{warning 'Eigenschaftenimplementierung hinzufügen'}
PROPERTY P_SpeedInPercent : LREAL
GET
P_SpeedInPercent := THIS^.rSpeedInPercentToSet;
END_GET
END_PROPERTY

PROPERTY P_StrokeLength : REAL
GET
P_StrokeLength := THIS^.rStrokeLength;
END_GET
END_PROPERTY

{warning 'Eigenschaftenimplementierung hinzufügen'}
PROPERTY P_StrokeLengthInitialized : BOOL
GET
P_StrokeLengthInitialized := THIS^.bStrokeLengthInitialized;
END_GET
SET
THIS^.bStrokeLengthInitialized := P_StrokeLengthInitialized;
END_SET
END_PROPERTY

PROPERTY P_WorkPressure : REAL
GET
P_WorkPressure := THIS^.rCurrentPressureInBar;
END_GET
END_PROPERTY

END_FUNCTION_BLOCK

(* stored: Version 1.1.0.1, ProductVersion 3.1.4024.12
   POU FB_CYLINDER_DA_TESTDEV1: Id {869475c7-ef97-4a7c-8ba5-1a42b23da02a}, SpecialFunc None
   Folder PRIVAT: Id {5831127a-e495-46f5-8a0f-1d046bc33d11}
   Folder SEQUENCE: Id {a9bffe34-56d4-42a0-bd85-2120cfcc493b}
   Method _m_DebugManager: Id {3c0314c9-f958-4098-88b9-d633cb92bde6}
   Method _m_Delay: Id {4de8ce80-6b9e-428f-9ea5-2ff018cbca80}
   Method _m_GeneralStepSetting: Id {24d8fd13-b379-4769-a659-85f3a480beb1}
   Method _m_HMI: Id {f56e0455-8f05-427d-ae10-35ce3dd7ec48}
   Method _m_ManualOperation: Id {08ef6f8c-9fc2-4a0c-ad9f-9f46c3bbc957}
   Method _m_PressureCalibration: Id {34794bd8-8f30-4a1c-bded-6683db0c4b4c}
   Method _m_PressureRegulation: Id {b0e232cf-6ed7-46e2-900f-075612c3a0f9}
   Method _m_Recording: Id {df88b879-7071-4b2f-a597-6e80be8b9c71}
   Method _m_SaveLastStep: Id {9fdaa3b9-a96c-4bff-bb87-77a3e60df6bb}
   Method _m_Seq_INIT: Id {f9cfc93d-4b0f-43dd-ab42-c65811c2e031}
   Method _m_Seq_LOW_PRESSURE_CALIBRATION: Id {1318f128-dd64-4e95-89a0-884e121348f4}
   Method _m_Seq_LOW_PRESSURE_MODE: Id {f82ab1c7-c9ef-435d-9f8b-8c61489859a6}
   Method _m_Seq_OPEN_LOCK_VALVES: Id {b7cfbdb7-7d40-423e-8fff-728fd5186b1e}
   Method _m_Seq_OPEN_RESERVOIR: Id {e1236d95-c6e4-4c6f-a7f3-534cb4bf9b62}
   Method _m_Seq_PRESSURE_CALIBRATION: Id {1bfc6a85-663e-4024-8ab2-022a9e48ea16}
   Method _m_Seq_PUMP2_ADD: Id {1baeb679-c052-4be0-8a42-e0985d7a075e}
   Method _m_Seq_PUMP3_ADD: Id {91b2c056-8d1b-40bd-b9b4-ee7732a8764d}
   Method _m_Seq_PUMP4_ADD: Id {9f51ed93-3bb9-4a3d-8f66-c8bb58c50c06}
   Method _m_Seq_SET_MAX_POS: Id {a4ff45b1-09e0-4222-a355-b456c9816aeb}
   Method _m_Seq_SET_WORK_PRESSURE: Id {cc2c3b1d-434f-4870-918e-924ee5476c2f}
   Method _m_Seq_SET_ZERO_POS: Id {a0698914-5d1c-48f0-b6d0-ead3eebb9680}
   Method _m_Seq_STOP: Id {5a3e320f-112a-4844-b8ff-ad7e993876ce}
   Method _m_Seq_STOP_AND_LOCK: Id {d01e608a-17c4-4d36-a5d6-d8a44fccd4da}
   Method _m_Seq_TO_HP: Id {93cdc5d4-9ecd-488d-babb-0c1575d8e8d4}
   Method _m_Seq_TO_SET_POS: Id {2c0f225f-9b0a-4aae-b925-08b548f42d15}
   Method _m_Seq_TO_WP: Id {5ba5b69d-8d51-4ff0-a3ee-fd4a54b59f89}
   Method _m_SequenceManager: Id {a82c7186-75d7-41f9-a75c-fb34f442338a}
   Method _m_SpeedRegulation: Id {bde6a516-003e-4041-b299-332af2ff0a98}
   Method _m_TimeOut: Id {4d7a21df-4d0e-456e-837a-6e1ec028adba}
   Method FB_init: Id {3eddab45-6958-4dfd-8b24-1deffd8654a6}
   Method M_LowPressureCalibration: Id {4c4aa761-4ce6-4927-99ce-753ef2c83bac}
   Method M_LowPressureMode: Id {ffc0cadb-621c-44b9-8086-c56093a333f6}
   Method M_OpenLockValves: Id {9d7190d5-3e74-4fb9-954e-0504316da3b0}
   Method M_OpenReservoir: Id {4d05e67f-0bcd-4d4d-89ad-643ecfe61b4f}
   Method M_PressureCalibration: Id {95a02b1f-d857-4bb7-8e27-77402689bfbf}
   Method M_Pump2Add: Id {88f3a218-cc95-4bf0-b16d-163da42870b5}
   Method M_Pump3Add: Id {c24a4452-1376-4ce6-a3ab-19c9ec15d08e}
   Method M_Pump4Add: Id {75eda3be-013d-4e3a-b91d-bfd32528cd7a}
   Method M_Reset: Id {51185ceb-0608-4fb2-82ca-2fdc35a10112}
   Method M_Run: Id {23e5959b-1f76-44e9-b254-e7757dbd1b8c}
   Method M_SetMaxPos: Id {bb4d4dca-6123-4524-b431-23bb935eee74}
   Method M_SetReady: Id {d9e65538-b03d-4723-b24c-4503df9eaef2}
   Method M_SetWorkPressure: Id {b51b9fcf-a17a-49ed-b114-876c3efd1a1a}
   Method M_SetZeroPos: Id {3aad99c8-3b93-4b4c-95b9-950170a10e45}
   Method M_Stop: Id {49a98cb3-5742-4c81-97f6-41549c0a6194}
   Method M_StopAndLock: Id {f07563c3-75a4-4012-a26b-70e4e023623a}
   Method M_ToHP: Id {fe8cf06b-e261-4737-851b-dfa0a48b2569}
   Method M_ToSetPos: Id {44cdaf68-bebc-4b53-b732-e3d0c25a0570}
   Method M_ToWP: Id {42eccb49-e3a0-4f84-9df1-89e9492bac4f}
   Property P_ActiveDirection: Id {bb177c56-5bf4-456b-bd35-4110bf2c0b6b}
   Get Get: Id {81862fc7-8740-48d6-aabb-750d3f4aa01e}
   Property P_ActiveVolumeFlow: Id {946f3b6b-b04f-4592-a5d6-37e4a19507d5}
   Get Get: Id {abd0562a-6524-4426-82ad-461c174736ab}
   Property P_CurrentForceInKN: Id {6c649f8a-2cb9-4c53-a460-6728e479212a}
   Get Get: Id {3ee17635-3cb1-47d0-9298-d2a1694411b6}
   Property P_DoubleActing: Id {5d7ac27f-14e0-409a-ba97-dda6248a40da}
   Get Get: Id {0beebe25-6228-4f14-946f-52856e4bb06d}
   Property P_Event: Id {31da0ff1-1dfd-4e32-b8ac-0cb534ab2b59}
   Get Get: Id {ea8eb761-a1fb-4af3-8d9c-dc884b6aba71}
   Set Set: Id {eedfdc11-1201-44c7-91df-13c0241d5659}
   Property P_FullObjectPath: Id {f4b51499-f863-40ce-a072-20999b9fe9a3}
   Get Get: Id {5901c2fa-eda4-4d5d-8c4f-f4141c32c492}
   Set Set: Id {781f8bf3-4ce8-486b-b4b0-51206a6f96d2}
   Property P_Global_Ack: Id {d5036133-64f7-4f9e-a413-2f769fc7f207}
   Get Get: Id {84859d05-d51e-48f0-9b19-2a76ccc49b02}
   Set Set: Id {224b9ca1-1704-4d02-9c9f-2d98b2303f3e}
   Property P_GlobalID: Id {1f8794ac-59f7-4097-9335-26e805a10d87}
   Get Get: Id {0d8c0c77-d0ae-429b-a753-731140411ead}
   Property P_LowPressure: Id {8360123c-b111-49fc-8952-81201de0e957}
   Get Get: Id {f20bbd60-1f27-491c-b237-908a7d58ba07}
   Property P_LowPressureChA: Id {701b8f3f-ea17-4898-9856-3b520b81dd7e}
   Get Get: Id {ecdb97ab-3f8e-4a79-b663-74b2d1833e48}
   Property P_LowPressureChB: Id {8572c222-9080-4ca7-880d-9909692f2624}
   Get Get: Id {728077ee-e2ba-4ef8-99a2-da95007fc54c}
   Property P_LowPressureModeEnable: Id {1fe6839d-8940-4533-a401-c4cc583e6577}
   Get Get: Id {4e27dfa8-7aa6-4726-8e1e-1c44da369649}
   Property P_MaxPosVal: Id {cff043fe-ab6a-47f5-aa1a-c070fe6ac24e}
   Get Get: Id {c5fbf8f1-9ff5-46c4-aa5d-f85bafebb367}
   Property P_MinPosVal: Id {be0fed34-5310-407d-9569-733869df6eed}
   Get Get: Id {71627298-a9bf-4f85-b030-b5fd87ea4921}
   Property P_PistonSurfaceA: Id {d11e6507-3d7d-49ad-a78f-d26b44d8a120}
   Get Get: Id {02d08729-561d-4f23-b115-1be9657e05fb}
   Property P_PistonSurfaceB: Id {74ce623a-169e-4d05-99ff-2258345f7b39}
   Get Get: Id {0d425fd2-6cb5-4656-8829-7fbbb4b5d77a}
   Property P_Position: Id {50cea76f-aa4a-4d81-84a1-03e14ce2d44f}
   Get Get: Id {574a9eba-f8ef-4f68-8257-d8be892171f0}
   Property P_PositionAbs: Id {fb0c1f48-bc86-4e82-961e-58a1bdadf556}
   Get Get: Id {7559cd9f-553d-4c70-be31-9f3bcb98eb2d}
   Property P_PressureChA: Id {76819b6d-040f-44cb-8891-1d943fe769d3}
   Get Get: Id {405dc3a6-747c-44b0-b5ba-7646ac5ed9f9}
   Property P_PressureChB: Id {97943423-0d75-450c-b956-4f50df16d1d1}
   Get Get: Id {927e9357-7682-4ccf-bc34-5349f2db9ca3}
   Property P_PressureOk: Id {2de9a025-dc62-40fb-9172-cf58778bba7a}
   Get Get: Id {b333847b-c944-4d48-8ce8-334cd1ea9cc7}
   Property P_Pump2Added: Id {f8e8ef84-a094-4cc2-9421-ccce644f8ff9}
   Get Get: Id {482c7cbe-eb76-4d4d-8957-67f26dac2945}
   Property P_Pump3Added: Id {d4cbe0e5-c074-451b-8f66-ff7601c3b008}
   Get Get: Id {b46d9bf0-9177-417d-a2e1-6db0ced83b5f}
   Property P_Pump4Added: Id {7bcfda4d-94e1-4f7e-8c99-9e226f519c23}
   Get Get: Id {8a3d0f4a-6577-426e-bfc9-0f69605be178}
   Property P_ReadyState: Id {2350a514-d7c0-496b-a8a1-3d05b684b233}
   Get Get: Id {af5c0915-940c-49bd-b35e-7471c6df3a7f}
   Property P_ReservoirAOpened: Id {940b5819-d7b2-487a-8b30-9255d99dd3e8}
   Get Get: Id {e6007e89-9b37-4c19-a0cf-fbb55436dfdc}
   Property P_ReservoirBOpened: Id {748caa81-2fe4-4cb4-a8a4-b54b633b4eb4}
   Get Get: Id {5da4f544-4c9a-4ce0-bc86-09af2c4773ef}
   Property P_ReservoirPressure: Id {2df6ee14-4f4b-4a0a-9de8-4fa8896d4e9b}
   Get Get: Id {c7a4d39e-e506-47ae-b3da-4ab415575379}
   Property P_SpeedInMmPerSecond: Id {eb079ba1-a563-4e89-bf88-28dd55805810}
   Get Get: Id {771dab11-7c62-46aa-ab12-667b088cf5cc}
   Property P_SpeedInPercent: Id {3f2beb92-2ba2-455d-8a2e-96a82bccf2d6}
   Get Get: Id {85c814c3-2a54-4cf4-9799-1a8b52edf644}
   Property P_StrokeLength: Id {fbaf65dd-42cb-4f8d-8f49-8c8def1cadbf}
   Get Get: Id {b8dbf7f9-e521-4e20-9359-c0e1ea5a4686}
   Property P_StrokeLengthInitialized: Id {9b9b22c3-e42e-4294-bd56-8508070dcfd8}
   Get Get: Id {31db4f29-c0a4-4fe4-904e-86c2cfd2ba66}
   Set Set: Id {c5086115-0405-4eeb-9c0f-edce1d4afb0b}
   Property P_WorkPressure: Id {296bb44d-e73b-4a3a-8282-54e3e52b2e97}
   Get Get: Id {a2602ed8-eeab-44e2-a19a-4298301a6382} *)
